Yaskawa INFORM job: demo_21_12_2023_planes_program.JBI

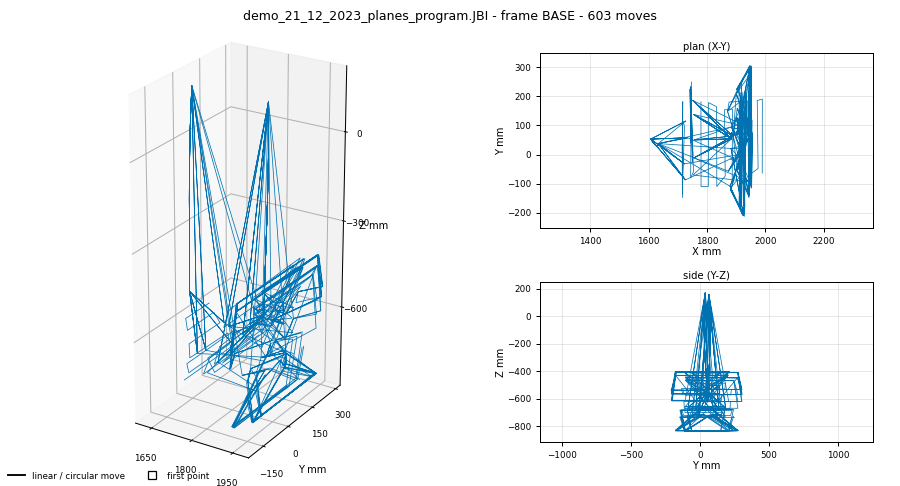
[picture p0: tool path of demo_21_12_2023_planes_program.JBI in frame BASE, 603 of 622 moves have a stored position in this frame; points joined in program order, loops and branches not executed]
/JOB
//NAME demo_21_12_2023_planes_program
//POS
///NPOS 616,0,616,0,0,0
///TOOL 0
///POSTYPE BASE
///RECTAN
///RCONF 0,0,0,0,0,0,0,0,0,0,0,0,0,0,0,0,0,0,0,0,0,0,0,0
C00000=1907.033318,105.448562,-531.357100,175.000000,-89.559174,-5.000000
C00001=1954.483034,118.521309,-531.351102,-175.000000,-89.985238,-46.086947
C00002=1951.789589,-60.582177,-405.692341,-175.000000,-58.956246,33.554175
C00003=1950.891473,275.514781,-409.751002,175.000000,-60.779903,-37.214964
C00004=1950.739483,304.407695,-531.280759,-175.000000,-89.985238,-46.086947
C00005=1904.555206,228.496419,-531.310537,175.000000,-9000000,5.000000
C00006=1955.420788,71.957040,-531.368723,175.000000,-89.985238,-46.086947
C00007=1952.438991,-107.141483,-443.395354,175.000000,-58.956472,33.555545
C00008=1950.674715,271.761571,-447.437042,-175.000000,-60.779789,-37.213566
C00009=1950.815178,300.649067,-531.282181,175.000000,-89.985238,-46.086947
C00010=1904.555206,228.496419,-531.310537,175.000000,-9000000,5.000000
C00011=1955.560862,65.001669,-531.371355,175.000000,-89.985238,-46.086947
C00012=1952.862971,-114.102374,-406.302816,-175.000000,-58.956353,33.554309
C00013=1950.927845,273.475107,-410.342085,175.000000,-60.780048,-37.215010
C00014=1950.780573,302.367348,-531.281531,175.000000,-89.985238,-46.086947
C00015=1904.555206,228.496419,-531.310537,175.000000,-9000000,5.000000
C00016=1900.400389,222.474608,-568.500057,175.000000,-89.559174,-5.000000
C00017=1947.081445,305.285270,-568.478734,-175.000000,-89.990197,-46.567779
C00018=1947.250662,275.979199,-409.311487,175.000000,-60.601810,-37.547371
C00019=1943.764744,-60.153943,-406.108555,175.000000,-59.166964,33.242469
C00020=1947.704549,119.398883,-568.525070,175.000000,-89.990197,-46.567779
C00021=1900.913317,69.456215,-568.538199,175.000000,-9000000,5.000000
C00022=1947.094044,301.526641,-568.479671,175.000000,-89.990197,-46.567779
C00023=1946.974018,272.228543,-446.996811,175.000000,-60.601591,-37.547423
C00024=1943.630528,-106.710862,-443.805636,175.000000,-59.167227,33.242548
C00025=1947.860635,72.834614,-568.536677,175.000000,-89.990197,-46.567779
C00026=1900.913317,69.456215,-568.538199,175.000000,-9000000,5.000000
C00027=1947.088284,303.244923,-568.479242,-175.000000,-89.990197,-46.567779
C00028=1947.253324,273.939620,-409.902004,-175.000000,-60.601821,-37.547527
C00029=1943.938758,-113.673732,-406.712292,175.000000,-59.167149,33.242355
C00030=1947.883950,65.879243,-568.538410,175.000000,-89.990197,-46.567779
C00031=1900.913317,69.456215,-568.538199,175.000000,-9000000,5.000000
C00032=1947.181211,275.522780,-568.486153,175.000000,-89.990197,-46.567779
C00033=1946.900224,246.230934,-467.867787,175.000000,-60.602079,-37.547614
C00034=1943.466507,-105.922888,-464.668327,175.000000,-59.167008,33.241936
C00035=1947.858017,73.615805,-568.536482,175.000000,-89.990197,-46.567779
C00036=1900.913317,69.456215,-568.538199,175.000000,-9000000,5.000000
C00037=1889.556234,63.921597,158.246462,-12.170215,-10.697646,-175.000000
C00038=1889.623159,63.877828,158.302867,-12.170828,-10.698957,-175.000000
C00039=1887.716063,68.814383,78.786651,-10.416760,-13.956672,-175.000000
C00040=1886.079895,71.876277,1.464639,-8.880031,-17.287043,-175.000000
C00041=1884.307478,73.313181,-73.802853,-7.558614,-20.681301,-175.000000
C00042=1882.911392,73.396272,-147.225748,-6.476440,-24.117963,-175.000000
C00043=1881.789821,72.259721,-218.453619,-5.660340,-27.576620,-175.000000
C00044=1880.837059,70.160415,-287.739273,5.000000,-31.424829,172.739336
C00045=1880.593414,67.184315,-355.151365,5.000000,-34.810443,174.015393
C00046=1880.906153,63.376292,-421.003543,5.000000,-38.223195,174.604447
C00047=1881.751155,59.024234,-485.031840,5.000000,-41.626153,174.627532
C00048=1883.567861,53.969547,-547.634242,5.000000,-44.999700,174.201251
C00049=1755.822095,50.404704,-618.581704,175.000000,-9000000,5.000000
C00050=1889.556234,63.921597,158.246462,-12.170215,-10.697646,-175.000000
C00051=1889.623159,63.877828,158.302867,-12.170828,-10.698957,-175.000000
C00052=1887.716063,68.814383,78.786651,-10.416760,-13.956672,-175.000000
C00053=1886.079895,71.876277,1.464639,-8.880031,-17.287043,-175.000000
C00054=1884.307478,73.313181,-73.802853,-7.558614,-20.681301,-175.000000
C00055=1882.911392,73.396272,-147.225748,-6.476440,-24.117963,-175.000000
C00056=1881.789821,72.259721,-218.453619,-5.660340,-27.576620,-175.000000
C00057=1880.837059,70.160415,-287.739273,5.000000,-31.424829,172.739336
C00058=1880.593414,67.184315,-355.151365,5.000000,-34.810443,174.015393
C00059=1880.906153,63.376292,-421.003543,5.000000,-38.223195,174.604447
C00060=1881.751155,59.024234,-485.031840,5.000000,-41.626153,174.627532
C00061=1883.567861,53.969547,-547.634242,5.000000,-44.999700,174.201251
C00062=1755.822095,50.404704,-618.581704,175.000000,-9000000,5.000000
C00063=1889.556234,63.921597,158.246462,-12.170215,-10.697646,-175.000000
C00064=1889.623159,63.877828,158.302867,-12.170828,-10.698957,-175.000000
C00065=1887.716063,68.814383,78.786651,-10.416760,-13.956672,-175.000000
C00066=1886.079895,71.876277,1.464639,-8.880031,-17.287043,-175.000000
C00067=1884.307478,73.313181,-73.802853,-7.558614,-20.681301,-175.000000
C00068=1882.911392,73.396272,-147.225748,-6.476440,-24.117963,-175.000000
C00069=1881.789821,72.259721,-218.453619,-5.660340,-27.576620,-175.000000
C00070=1880.837059,70.160415,-287.739273,5.000000,-31.424829,172.739336
C00071=1880.593414,67.184315,-355.151365,5.000000,-34.810443,174.015393
C00072=1880.906153,63.376292,-421.003543,5.000000,-38.223195,174.604447
C00073=1881.751155,59.024234,-485.031840,5.000000,-41.626153,174.627532
C00074=1883.567861,53.969547,-547.634242,5.000000,-44.999700,174.201251
C00075=1755.822095,50.404704,-618.581704,175.000000,-9000000,5.000000
C00076=1951.369555,117.933153,-618.544705,175.000000,-89.981843,-45.753303
C00077=1950.408580,-60.871163,-405.345417,-175.000000,-58.807688,33.768810
C00078=1946.465369,275.184802,-409.998652,175.000000,-60.901627,-36.982641
C00079=1945.459620,303.819540,-618.457694,175.000000,-89.981843,-45.753303
C00080=1900.287093,207.836706,-618.503937,175.000000,-9000000,5.000000
C00081=1952.849985,71.368885,-618.566501,175.000000,-89.981843,-45.753303
C00082=1951.598144,-107.427747,-443.052619,175.000000,-58.807922,33.768719
C00083=1946.295789,271.434354,-447.684920,175.000000,-60.901461,-36.982782
C00084=1945.579119,30060912,-618.459453,-175.000000,-89.981843,-45.753303
C00085=1900.287093,207.836706,-618.503937,175.000000,-9000000,5.000000
C00086=1953.071119,64.413513,-618.569757,-175.000000,-89.981843,-45.753303
C00087=1952.104538,-114.390894,-405.960815,175.000000,-58.807853,33.768670
C00088=1946.526026,273.145173,-410.589561,175.000000,-60.901614,-36.982778
C00089=1945.524489,301.779193,-618.458649,-175.000000,-89.981843,-45.753303
C00090=1900.287093,207.836706,-618.503937,175.000000,-9000000,5.000000
C00091=1952.825149,72.150076,-618.566135,-175.000000,-89.981843,-45.753303
C00092=1951.412479,-106.640599,-463.915398,175.000000,-58.807817,33.768501
C00093=1946.962416,245.436524,-468.560719,-175.000000,-60.901568,-36.983014
C00094=1946.405867,274.057050,-618.471626,175.000000,-89.981843,-45.753303
C00095=1900.287093,207.836706,-618.503937,175.000000,-9000000,5.000000
C00096=1889.556234,63.921597,158.246462,-12.170215,-10.697646,-175.000000
C00097=1889.623159,63.877828,158.302867,-12.170828,-10.698957,-175.000000
C00098=1887.716063,68.814383,78.786651,-10.416760,-13.956672,-175.000000
C00099=1886.079895,71.876277,1.464639,-8.880031,-17.287043,-175.000000
C00100=1884.307478,73.313181,-73.802853,-7.558614,-20.681301,-175.000000
C00101=1882.911392,73.396272,-147.225748,-6.476440,-24.117963,-175.000000
C00102=1881.789821,72.259721,-218.453619,-5.660340,-27.576620,-175.000000
C00103=1880.837059,70.160415,-287.739273,5.000000,-31.424829,172.739336
C00104=1880.593414,67.184315,-355.151365,5.000000,-34.810443,174.015393
C00105=1880.906153,63.376292,-421.003543,5.000000,-38.223195,174.604447
C00106=1881.751155,59.024234,-485.031840,5.000000,-41.626153,174.627532
C00107=1883.567861,53.969547,-547.634242,5.000000,-44.999700,174.201251
C00108=1750.649215,186.057193,-668.513072,175.000000,-9000000,5.000000
C00109=1889.556234,63.921597,158.246462,-12.170215,-10.697646,-175.000000
C00110=1889.623159,63.877828,158.302867,-12.170828,-10.698957,-175.000000
C00111=1887.716063,68.814383,78.786651,-10.416760,-13.956672,-175.000000
C00112=1886.079895,71.876277,1.464639,-8.880031,-17.287043,-175.000000
C00113=1884.307478,73.313181,-73.802853,-7.558614,-20.681301,-175.000000
C00114=1882.911392,73.396272,-147.225748,-6.476440,-24.117963,-175.000000
C00115=1881.789821,72.259721,-218.453619,-5.660340,-27.576620,-175.000000
C00116=1880.837059,70.160415,-287.739273,5.000000,-31.424829,172.739336
C00117=1880.593414,67.184315,-355.151365,5.000000,-34.810443,174.015393
C00118=1880.906153,63.376292,-421.003543,5.000000,-38.223195,174.604447
C00119=1881.751155,59.024234,-485.031840,5.000000,-41.626153,174.627532
C00120=1883.567861,53.969547,-547.634242,5.000000,-44.999700,174.201251
C00121=1750.649215,186.057193,-668.513072,175.000000,-9000000,5.000000
C00122=1889.556234,63.921597,158.246462,-12.170215,-10.697646,-175.000000
C00123=1889.623159,63.877828,158.302867,-12.170828,-10.698957,-175.000000
C00124=1887.716063,68.814383,78.786651,-10.416760,-13.956672,-175.000000
C00125=1886.079895,71.876277,1.464639,-8.880031,-17.287043,-175.000000
C00126=1884.307478,73.313181,-73.802853,-7.558614,-20.681301,-175.000000
C00127=1882.911392,73.396272,-147.225748,-6.476440,-24.117963,-175.000000
C00128=1881.789821,72.259721,-218.453619,-5.660340,-27.576620,-175.000000
C00129=1880.837059,70.160415,-287.739273,5.000000,-31.424829,172.739336
C00130=1880.593414,67.184315,-355.151365,5.000000,-34.810443,174.015393
C00131=1880.906153,63.376292,-421.003543,5.000000,-38.223195,174.604447
C00132=1881.751155,59.024234,-485.031840,5.000000,-41.626153,174.627532
C00133=1883.567861,53.969547,-547.634242,5.000000,-44.999700,174.201251
C00134=1750.649215,186.057193,-668.513072,175.000000,-9000000,5.000000
C00135=1941.739433,91.872264,-668.550173,5.000000,-89.981105,-135.836022
C00136=1942.819913,274.976952,-83002340,5.000000,-61.062899,143.242003
C00137=1946.018919,-60.273090,-834.731809,5.000000,-59.014144,-146.590892
C00138=1947.112174,-94.014122,-668.633050,5.000000,-89.981105,-135.836022
C00139=1905.452963,2.399975,-668.591073,175.000000,-9000000,5.000000
C00140=1941.848070,88.113636,-668.551849,5.000000,-89.981105,-135.836022
C00141=1945.998331,271.516439,-447.613467,175.000000,-60.871590,-37.040266
C00142=1950.423675,-107.356915,-443.127134,175.000000,-58.844853,33.715766
C00143=1951.553207,71.531040,-668.559002,-175.000000,-89.982681,-45.836017
C00144=1905.452963,2.399975,-668.591073,175.000000,-9000000,5.000000
C00145=1941.798406,89.831917,-668.551082,5.000000,-89.981105,-135.836022
C00146=1942.883974,272.936882,-829.346203,5.000000,-61.062928,143.241973
C00147=1947.570821,-113.793308,-834.098604,-5.000000,-59.014182,-146.590868
C00148=1951.754240,64.575669,-668.562103,-175.000000,-89.982681,-45.836017
C00149=1905.452963,2.399975,-668.591073,175.000000,-9000000,5.000000
C00150=1945.694838,274.219206,-668.468633,-175.000000,-89.982681,-45.836017
C00151=1946.589980,245.518494,-468.488538,-175.000000,-60.871631,-37.040464
C00152=1950.239929,-106.569854,-463.990120,175.000000,-58.844834,33.715560
C00153=1951.530628,72.312231,-668.558654,-175.000000,-89.982681,-45.836017
C00154=1905.452963,2.399975,-668.591073,175.000000,-9000000,5.000000
C00155=1889.556234,63.921597,158.246462,-12.170215,-10.697646,-175.000000
C00156=1889.623159,63.877828,158.302867,-12.170828,-10.698957,-175.000000
C00157=1887.716063,68.814383,78.786651,-10.416760,-13.956672,-175.000000
C00158=1886.079895,71.876277,1.464639,-8.880031,-17.287043,-175.000000
C00159=1884.307478,73.313181,-73.802853,-7.558614,-20.681301,-175.000000
C00160=1882.911392,73.396272,-147.225748,-6.476440,-24.117963,-175.000000
C00161=1881.789821,72.259721,-218.453619,-5.660340,-27.576620,-175.000000
C00162=1880.837059,70.160415,-287.739273,5.000000,-31.424829,172.739336
C00163=1880.593414,67.184315,-355.151365,5.000000,-34.810443,174.015393
C00164=1880.906153,63.376292,-421.003543,5.000000,-38.223195,174.604447
C00165=1881.751155,59.024234,-485.031840,5.000000,-41.626153,174.627532
C00166=1883.567861,53.969547,-547.634242,5.000000,-44.999700,174.201251
C00167=1754.643051,-11.429649,-718.589414,175.000000,-9000000,5.000000
C00168=1889.556234,63.921597,158.246462,-12.170215,-10.697646,-175.000000
C00169=1889.623159,63.877828,158.302867,-12.170828,-10.698957,-175.000000
C00170=1887.716063,68.814383,78.786651,-10.416760,-13.956672,-175.000000
C00171=1886.079895,71.876277,1.464639,-8.880031,-17.287043,-175.000000
C00172=1884.307478,73.313181,-73.802853,-7.558614,-20.681301,-175.000000
C00173=1882.911392,73.396272,-147.225748,-6.476440,-24.117963,-175.000000
C00174=1881.789821,72.259721,-218.453619,-5.660340,-27.576620,-175.000000
C00175=1880.837059,70.160415,-287.739273,5.000000,-31.424829,172.739336
C00176=1880.593414,67.184315,-355.151365,5.000000,-34.810443,174.015393
C00177=1880.906153,63.376292,-421.003543,5.000000,-38.223195,174.604447
C00178=1881.751155,59.024234,-485.031840,5.000000,-41.626153,174.627532
C00179=1883.567861,53.969547,-547.634242,5.000000,-44.999700,174.201251
C00180=1754.643051,-11.429649,-718.589414,175.000000,-9000000,5.000000
C00181=1889.556234,63.921597,158.246462,-12.170215,-10.697646,-175.000000
C00182=1889.623159,63.877828,158.302867,-12.170828,-10.698957,-175.000000
C00183=1887.716063,68.814383,78.786651,-10.416760,-13.956672,-175.000000
C00184=1886.079895,71.876277,1.464639,-8.880031,-17.287043,-175.000000
C00185=1884.307478,73.313181,-73.802853,-7.558614,-20.681301,-175.000000
C00186=1882.911392,73.396272,-147.225748,-6.476440,-24.117963,-175.000000
C00187=1881.789821,72.259721,-218.453619,-5.660340,-27.576620,-175.000000
C00188=1880.837059,70.160415,-287.739273,5.000000,-31.424829,172.739336
C00189=1880.593414,67.184315,-355.151365,5.000000,-34.810443,174.015393
C00190=1880.906153,63.376292,-421.003543,5.000000,-38.223195,174.604447
C00191=1881.751155,59.024234,-485.031840,5.000000,-41.626153,174.627532
C00192=1883.567861,53.969547,-547.634242,5.000000,-44.999700,174.201251
C00193=1754.643051,-11.429649,-718.589414,175.000000,-9000000,5.000000
C00194=1945.109419,-92.763747,-718.608360,5.000000,-89.988712,-136.492236
C00195=1944.744831,-59.705754,-834.062988,5.000000,-59.310215,-147.008189
C00196=1947.521106,275.607521,-830.600257,5.000000,-60.814495,142.793100
C00197=1943.996119,93.122640,-718.558252,5.000000,-89.988712,-136.492236
C00198=1903.328616,157.105618,-718.541637,175.000000,-9000000,5.000000
C00199=1950.912528,72.732070,-718.563642,-175.000000,-89.989413,-46.492234
C00200=1945.018194,-106.270873,-834.806367,-5.000000,-59.310282,-147.008065
C00201=1947.537237,271.848413,-831.332199,5.000000,-60.814515,142.793257
C00202=1944.018630,89.364012,-718.559266,-5.000000,-89.988712,-136.492236
C00203=1903.328616,157.105618,-718.541637,175.000000,-9000000,5.000000
C00204=1950.954184,65.776698,-718.565517,175.000000,-89.989413,-46.492234
C00205=1945.069512,-113.225825,-833.420115,5.000000,-59.310354,-147.008282
C00206=1947.538175,273.567484,-829.943731,5.000000,-60.814536,142.793056
C00207=1944.008339,91.082293,-718.558802,5.000000,-89.988712,-136.492236
C00208=1903.328616,157.105618,-718.541637,175.000000,-9000000,5.000000
C00209=1950.907849,73.513261,-718.563432,-175.000000,-89.989413,-46.492234
C00210=1945.021973,-105.488764,-833.644297,5.000000,-59.310234,-147.008242
C00211=1947.702278,245.845502,-830.177084,5.000000,-60.814585,142.793096
C00212=1944.174371,63.360150,-718.566275,5.000000,-89.988712,-136.492236
C00213=1903.328616,157.105618,-718.541637,175.000000,-9000000,5.000000
C00214=1889.556234,63.921597,158.246462,-12.170215,-10.697646,-175.000000
C00215=1889.623159,63.877828,158.302867,-12.170828,-10.698957,-175.000000
C00216=1887.716063,68.814383,78.786651,-10.416760,-13.956672,-175.000000
C00217=1886.079895,71.876277,1.464639,-8.880031,-17.287043,-175.000000
C00218=1884.307478,73.313181,-73.802853,-7.558614,-20.681301,-175.000000
C00219=1882.911392,73.396272,-147.225748,-6.476440,-24.117963,-175.000000
C00220=1881.789821,72.259721,-218.453619,-5.660340,-27.576620,-175.000000
C00221=1880.837059,70.160415,-287.739273,5.000000,-31.424829,172.739336
C00222=1880.593414,67.184315,-355.151365,5.000000,-34.810443,174.015393
C00223=1880.906153,63.376292,-421.003543,5.000000,-38.223195,174.604447
C00224=1881.751155,59.024234,-485.031840,5.000000,-41.626153,174.627532
C00225=1883.567861,53.969547,-547.634242,5.000000,-44.999700,174.201251
C00226=1754.303875,137.531750,-681.952455,175.000000,-9000000,5.000000
C00227=1889.556234,63.921597,158.246462,-12.170215,-10.697646,-175.000000
C00228=1889.623159,63.877828,158.302867,-12.170828,-10.698957,-175.000000
C00229=1887.716063,68.814383,78.786651,-10.416760,-13.956672,-175.000000
C00230=1886.079895,71.876277,1.464639,-8.880031,-17.287043,-175.000000
C00231=1884.307478,73.313181,-73.802853,-7.558614,-20.681301,-175.000000
C00232=1882.911392,73.396272,-147.225748,-6.476440,-24.117963,-175.000000
C00233=1881.789821,72.259721,-218.453619,-5.660340,-27.576620,-175.000000
C00234=1880.837059,70.160415,-287.739273,5.000000,-31.424829,172.739336
C00235=1880.593414,67.184315,-355.151365,5.000000,-34.810443,174.015393
C00236=1880.906153,63.376292,-421.003543,5.000000,-38.223195,174.604447
C00237=1881.751155,59.024234,-485.031840,5.000000,-41.626153,174.627532
C00238=1883.567861,53.969547,-547.634242,5.000000,-44.999700,174.201251
C00239=1754.303875,137.531750,-681.952455,175.000000,-9000000,5.000000
C00240=1889.556234,63.921597,158.246462,-12.170215,-10.697646,-175.000000
C00241=1889.623159,63.877828,158.302867,-12.170828,-10.698957,-175.000000
C00242=1887.716063,68.814383,78.786651,-10.416760,-13.956672,-175.000000
C00243=1886.079895,71.876277,1.464639,-8.880031,-17.287043,-175.000000
C00244=1884.307478,73.313181,-73.802853,-7.558614,-20.681301,-175.000000
C00245=1882.911392,73.396272,-147.225748,-6.476440,-24.117963,-175.000000
C00246=1881.789821,72.259721,-218.453619,-5.660340,-27.576620,-175.000000
C00247=1880.837059,70.160415,-287.739273,5.000000,-31.424829,172.739336
C00248=1880.593414,67.184315,-355.151365,5.000000,-34.810443,174.015393
C00249=1880.906153,63.376292,-421.003543,5.000000,-38.223195,174.604447
C00250=1881.751155,59.024234,-485.031840,5.000000,-41.626153,174.627532
C00251=1883.567861,53.969547,-547.634242,5.000000,-44.999700,174.201251
C00252=1754.303875,137.531750,-681.952455,175.000000,-9000000,5.000000
C00253=1889.556234,63.921597,158.246462,-12.170215,-10.697646,-175.000000
C00254=1889.623159,63.877828,158.302867,-12.170828,-10.698957,-175.000000
C00255=1887.716063,68.814383,78.786651,-10.416760,-13.956672,-175.000000
C00256=1886.079895,71.876277,1.464639,-8.880031,-17.287043,-175.000000
C00257=1884.307478,73.313181,-73.802853,-7.558614,-20.681301,-175.000000
C00258=1882.911392,73.396272,-147.225748,-6.476440,-24.117963,-175.000000
C00259=1881.789821,72.259721,-218.453619,-5.660340,-27.576620,-175.000000
C00260=1880.837059,70.160415,-287.739273,5.000000,-31.424829,172.739336
C00261=1880.593414,67.184315,-355.151365,5.000000,-34.810443,174.015393
C00262=1880.906153,63.376292,-421.003543,5.000000,-38.223195,174.604447
C00263=1881.751155,59.024234,-485.031840,5.000000,-41.626153,174.627532
C00264=1883.567861,53.969547,-547.634242,5.000000,-44.999700,174.201251
C00265=1754.303875,137.531750,-681.952455,175.000000,-9000000,5.000000
C00266=1944.740157,93.554557,-681.959370,-5.000000,-89.991235,-136.713417
C00267=1949.343284,275.815144,-830.807048,5.000000,-60.729125,142.642519
C00268=1944.552036,-59.508291,-833.842699,-5.000000,-59.408325,-147.150251
C00269=1944.418269,-92.331830,-681.998435,5.000000,-89.991235,-136.713417
C00270=1903.729498,-56.819837,-681.991470,175.000000,-9000000,5.000000
C00271=1944.733648,89.795928,-681.960160,5.000000,-89.991235,-136.713417
C00272=1949.330371,272.055939,-831.538811,5.000000,-60.729126,142.642723
C00273=1944.465133,-106.073368,-834.582953,5.000000,-59.408549,-147.150209
C00274=1944.337637,-138.896099,-682.008221,5.000000,-89.991235,-136.713417
C00275=1903.729498,-56.819837,-681.991470,175.000000,-9000000,5.000000
C00276=1944.736623,91.514210,-681.959798,5.000000,-89.991235,-136.713417
C00277=1949.344074,273.774978,-830.150143,5.000000,-60.729278,142.642595
C00278=1944.463820,-113.028499,-833.196650,-5.000000,-59.408464,-147.150271
C00279=1944.325592,-145.851470,-682.009683,-5.000000,-89.991235,-136.713417
C00280=1903.729498,-56.819837,-681.991470,175.000000,-9000000,5.000000
C00281=1944.688619,63.792067,-681.965625,5.000000,-89.991235,-136.713417
C00282=1949.294155,246.053003,-830.381801,5.000000,-60.729348,142.642640
C00283=1944.476511,-105.291509,-833.421558,-5.000000,-59.408226,-147.150148
C00284=1944.338989,-138.114908,-682.008057,-5.000000,-89.991235,-136.713417
C00285=1903.729498,-56.819837,-681.991470,175.000000,-9000000,5.000000
C00286=1889.556234,63.921597,158.246462,-12.170215,-10.697646,-175.000000
C00287=1889.623159,63.877828,158.302867,-12.170828,-10.698957,-175.000000
C00288=1887.716063,68.814383,78.786651,-10.416760,-13.956672,-175.000000
C00289=1886.079895,71.876277,1.464639,-8.880031,-17.287043,-175.000000
C00290=1884.307478,73.313181,-73.802853,-7.558614,-20.681301,-175.000000
C00291=1882.911392,73.396272,-147.225748,-6.476440,-24.117963,-175.000000
C00292=1881.789821,72.259721,-218.453619,-5.660340,-27.576620,-175.000000
C00293=1880.837059,70.160415,-287.739273,5.000000,-31.424829,172.739336
C00294=1880.593414,67.184315,-355.151365,5.000000,-34.810443,174.015393
C00295=1880.906153,63.376292,-421.003543,5.000000,-38.223195,174.604447
C00296=1881.751155,59.024234,-485.031840,5.000000,-41.626153,174.627532
C00297=1883.567861,53.969547,-547.634242,5.000000,-44.999700,174.201251
C00298=1752.029754,-69.858282,-731.982788,175.000000,-9000000,5.000000
C00299=1942.290332,-92.571429,-731.985649,5.000000,-89.989735,-136.581685
C00300=1942.741090,-59.625904,-833.959304,5.000000,-59.349806,-147.065680
C00301=1946.332931,275.692102,-830.669243,5.000000,-60.779904,142.731914
C00302=1941.757450,93.314957,-731.940007,5.000000,-89.989735,-136.581685
C00303=1901.186698,127.297726,-731.932241,175.000000,-9000000,5.000000
C00304=1942.423818,-139.135698,-731.997082,-5.000000,-89.989735,-136.581685
C00305=1942.867588,-106.191308,-834.700067,5.000000,-59.350536,-147.065659
C00306=1946.336088,271.931920,-831.400871,5.000000,-60.780021,142.732704
C00307=1941.768225,89.556329,-731.940930,5.000000,-89.989735,-136.581685
C00308=1901.186698,127.297726,-731.932241,175.000000,-9000000,5.000000
C00309=1942.443758,-146.091069,-731.998790,5.000000,-89.989735,-136.581685
C00310=1942.898325,-113.146105,-833.314387,5.000000,-59.350283,-147.065833
C00311=1946.341642,273.651504,-83011340,-5.000000,-60.780524,142.732427
C00312=1941.763299,91.274610,-731.940508,5.000000,-89.989735,-136.581685
C00313=1901.186698,127.297726,-731.932241,175.000000,-9000000,5.000000
C00314=1942.421579,-138.354507,-731.996890,5.000000,-89.989735,-136.581685
C00315=1942.874857,-105.408541,-833.539318,5.000000,-59.349912,-147.065963
C00316=1946.420644,245.930307,-830.244454,5.000000,-60.780388,142.731955
C00317=1941.842770,63.552467,-731.947315,5.000000,-89.989735,-136.581685
C00318=1901.186698,127.297726,-731.932241,18000000,-6000000,000000
C00319=1744.163168,103.731386,-533.824639,5.000000,-89.520571,175.000000
C00320=174053701,229.900913,-533.872980,5.000000,-89.520571,175.000000
C00321=1740.139661,223.998415,-571.035053,5.000000,-89.520571,175.000000
C00322=1745.940022,70.141244,-570.969500,5.000000,-89.520571,175.000000
C00323=1743.699231,39.699755,-620.986636,5.000000,-89.520571,175.000000
C00324=1743.736408,220.431312,-621.006311,5.000000,-89.520571,175.000000
C00325=1743.938875,217.744936,-671.006071,5.000000,-89.520571,175.000000
C00326=1751.483237,3.541384,-670.919251,5.000000,-89.520571,175.000000
C00327=1749.639439,-25.239911,-720.933248,5.000000,-89.520571,175.000000
C00328=1742.908909,221.089212,-721.016811,5.000000,-89.520571,175.000000
C00329=1744.116223,233.211429,-684.407259,5.000000,-89.520571,175.000000
C00330=1753.513039,-58.753955,-684.296338,5.000000,-89.520571,175.000000
C00331=1743.842593,-79.925565,-734.376670,5.000000,-89.520571,175.000000
C00332=1746.666835,248.969851,-734.389409,18000000,-6000000,000000
C00333=1717.090387,-3.043329,-525.112751,-5.000000,-89.896397,-175.000000
C00334=1715.582850,-134.626368,-525.110413,-5.000000,-89.896397,-175.000000
C00335=1715.652100,-125.400738,-569.935144,-5.000000,-89.896397,-175.000000
C00336=1714.677180,27.356629,-569.942784,-5.000000,-89.896397,-175.000000
C00337=1716.200893,60.962231,-619.941404,-5.000000,-89.896397,-175.000000
C00338=1715.751699,-117.347731,-619.935355,-5.000000,-89.896397,-175.000000
C00339=1715.928918,-113.952816,-669.935247,-5.000000,-89.896397,-175.000000
C00340=1722.693836,97.479027,-669.931151,-5.000000,-89.896397,-175.000000
C00341=1715.897617,118.196967,-719.944318,-5.000000,-89.896397,-175.000000
C00342=1715.387537,-119.836296,-719.936081,-5.000000,-89.896397,-175.000000
C00343=1715.633277,-131.036930,-683.332748,-5.000000,-89.896397,-175.000000
C00344=1716.169223,154.077841,-683.342749,-5.000000,-89.896397,-175.000000
C00345=1716.790282,181.476308,-733.342762,-5.000000,-89.896397,-175.000000
C00346=1716.082413,-146.810235,-733.331410,18000000,-6000000,000000
C00347=1878.651480,-14.855522,-537.062852,175.000000,-88.097363,-5.000000
C00348=1922.281376,-31.606783,-537.075471,5.000000,-89.970325,-133.774897
C00349=1921.565087,150.704793,-403.442618,-175.000000,-59.777968,-34.809520
C00350=193001845,-180.972615,-402.864288,175.000000,-59.463968,37.005505
C00351=1927.472959,-211.533153,-537.206326,5.000000,-89.970325,-133.774897
C00352=1881.720340,-121.213359,-537.140203,-175.000000,-89.999999,5.000000
C00353=1920.818604,19.088977,-537.038602,5.000000,-89.970325,-133.774897
C00354=1919.228609,201.394910,-429.719115,175.000000,-59.777914,-34.809652
C00355=1929.050258,-178.319874,-429.176665,-175.000000,-59.464338,37.005437
C00356=1927.396225,-208.873762,-537.204392,5.000000,-89.970325,-133.774897
C00357=1881.720340,-121.213359,-537.140203,-175.000000,-89.999999,5.000000
C00358=1920.513394,29.666722,-537.030909,5.000000,-89.970325,-133.774897
C00359=1919.781998,211.979285,-403.878868,-175.000000,-59.777995,-34.809835
C00360=1929.779916,-173.832647,-403.339775,175.000000,-59.463942,37.005472
C00361=1927.266945,-204.393259,-537.201133,5.000000,-89.970325,-133.774897
C00362=1881.720340,-121.213359,-537.140203,-175.000000,-89.999999,5.000000
C00363=1880.324864,-121.388096,-563.848788,175.000000,-88.097363,-5.000000
C00364=1924.477331,-209.309200,-563.788106,175.000000,-89.972614,45.007217
C00365=1928.547064,-179.814548,-403.922550,175.000000,-59.929655,36.165405
C00366=1930.987541,151.882666,-402.634194,-175.000000,-59.304595,-35.645060
C00367=1926.936425,-29.382830,-563.911404,-175.000000,-89.972614,45.007217
C00368=1882.272046,21.082740,-563.946419,-175.000000,-89.999999,5.000000
C00369=1924.513677,-206.649809,-563.789928,175.000000,-89.972614,45.007217
C00370=1927.708515,-177.161618,-430.238366,175.000000,-59.929885,36.165300
C00371=1930.807006,202.572899,-428.982251,175.000000,-59.304515,-35.645269
C00372=1927.629296,21.312930,-563.946144,-175.000000,-89.972614,45.007217
C00373=1882.272046,21.082740,-563.946419,-175.000000,-89.999999,5.000000
C00374=1924.574913,-202.169306,-563.792998,175.000000,-89.972614,45.007217
C00375=1928.629244,-172.674803,-404.407974,-175.000000,-59.929560,36.165524
C00376=1931.808346,213.156570,-403.157323,175.000000,-59.304780,-35.644990
C00377=1927.773864,31.890675,-563.953393,-175.000000,-89.972614,45.007217
C00378=1882.272046,21.082740,-563.946419,-175.000000,-89.999999,5.000000
C00379=1632.892026,37.747570,168.285511,11.376794,11.539120,-175.000000
C00380=1632.827507,37.791596,168.344749,11.377310,11.540473,-175.000000
C00381=1631.070965,33.437366,89.156599,9.359774,14.678599,-175.000000
C00382=1629.142714,30.961716,12.173907,7.532522,17.899912,-175.000000
C00383=1627.447598,30.112422,-62.761067,5.887863,21.196066,-175.000000
C00384=1625.471635,30.613173,-135.840164,5.000000,24.547751,-175.000000
C00385=1623.335953,32.324503,-206.720523,5.000000,27.937078,-175.000000
C00386=1621.140462,34.985091,-275.661674,5.000000,-31.424829,-5.000000
C00387=1618.347384,38.503638,-342.713252,5.000000,-34.810443,-5.000000
C00388=1615.097741,42.831038,-408.197316,-5.000000,-38.223195,-5.000000
C00389=1611.433002,47.673610,-471.854532,-5.000000,-41.626153,-5.000000
C00390=1606.899024,53.186011,-534.066843,5.000000,-44.999700,-5.000000
C00391=1733.759636,57.739172,-614.031896,-175.000000,-89.999999,5.000000
C00392=1632.892026,37.747570,168.285511,11.376794,11.539120,-175.000000
C00393=1632.827507,37.791596,168.344749,11.377310,11.540473,-175.000000
C00394=1631.070965,33.437366,89.156599,9.359774,14.678599,-175.000000
C00395=1629.142714,30.961716,12.173907,7.532522,17.899912,-175.000000
C00396=1627.447598,30.112422,-62.761067,5.887863,21.196066,-175.000000
C00397=1625.471635,30.613173,-135.840164,5.000000,24.547751,-175.000000
C00398=1623.335953,32.324503,-206.720523,5.000000,27.937078,-175.000000
C00399=1621.140462,34.985091,-275.661674,5.000000,-31.424829,-5.000000
C00400=1618.347384,38.503638,-342.713252,5.000000,-34.810443,-5.000000
C00401=1615.097741,42.831038,-408.197316,-5.000000,-38.223195,-5.000000
C00402=1611.433002,47.673610,-471.854532,-5.000000,-41.626153,-5.000000
C00403=1606.899024,53.186011,-534.066843,5.000000,-44.999700,-5.000000
C00404=1733.759636,57.739172,-614.031896,-175.000000,-89.999999,5.000000
C00405=1632.892026,37.747570,168.285511,11.376794,11.539120,-175.000000
C00406=1632.827507,37.791596,168.344749,11.377310,11.540473,-175.000000
C00407=1631.070965,33.437366,89.156599,9.359774,14.678599,-175.000000
C00408=1629.142714,30.961716,12.173907,7.532522,17.899912,-175.000000
C00409=1627.447598,30.112422,-62.761067,5.887863,21.196066,-175.000000
C00410=1625.471635,30.613173,-135.840164,5.000000,24.547751,-175.000000
C00411=1623.335953,32.324503,-206.720523,5.000000,27.937078,-175.000000
C00412=1621.140462,34.985091,-275.661674,5.000000,-31.424829,-5.000000
C00413=1618.347384,38.503638,-342.713252,5.000000,-34.810443,-5.000000
C00414=1615.097741,42.831038,-408.197316,-5.000000,-38.223195,-5.000000
C00415=1611.433002,47.673610,-471.854532,-5.000000,-41.626153,-5.000000
C00416=1606.899024,53.186011,-534.066843,5.000000,-44.999700,-5.000000
C00417=1733.759636,57.739172,-614.031896,-175.000000,-89.999999,5.000000
C00418=1927.328468,-28.623634,-613.927963,175.000000,-89.953719,44.592323
C00419=1934.355931,152.264475,-402.352265,175.000000,-59.137640,-35.925997
C00420=1928.209886,-179.401451,-404.276647,-175.000000,-6082734,35.875902
C00421=1922.262476,-208.550004,-613.718064,175.000000,-89.953719,44.592323
C00422=1879.006381,-108.476117,-613.835557,-175.000000,-89.999999,5.000000
C00423=1928.755854,22.072125,-613.987103,175.000000,-89.953719,44.592323
C00424=1934.908337,202.954235,-428.725120,175.000000,-59.137750,-35.925865
C00425=1927.410838,-176.748780,-430.593291,175.000000,-6082759,35.876024
C00426=1922.337354,-205.890613,-613.721167,-175.000000,-89.953719,44.592323
C00427=1879.006381,-108.476117,-613.835557,-175.000000,-89.999999,5.000000
C00428=1929.053680,32.649871,-613.999443,175.000000,-89.953719,44.592323
C00429=1936.065735,213.538641,-402.904501,175.000000,-59.137643,-35.926149
C00430=1928.394599,-172.261419,-404.765772,175.000000,-6082764,35.875812
C00431=1922.463506,-201.410110,-613.726394,175.000000,-89.953719,44.592323
C00432=1879.006381,-108.476117,-613.835557,-175.000000,-89.999999,5.000000
C00433=1632.892026,37.747570,168.285511,11.376794,11.539120,-175.000000
C00434=1632.827507,37.791596,168.344749,11.377310,11.540473,-175.000000
C00435=1631.070965,33.437366,89.156599,9.359774,14.678599,-175.000000
C00436=1629.142714,30.961716,12.173907,7.532522,17.899912,-175.000000
C00437=1627.447598,30.112422,-62.761067,5.887863,21.196066,-175.000000
C00438=1625.471635,30.613173,-135.840164,5.000000,24.547751,-175.000000
C00439=1623.335953,32.324503,-206.720523,5.000000,27.937078,-175.000000
C00440=1621.140462,34.985091,-275.661674,5.000000,-31.424829,-5.000000
C00441=1618.347384,38.503638,-342.713252,5.000000,-34.810443,-5.000000
C00442=1615.097741,42.831038,-408.197316,-5.000000,-38.223195,-5.000000
C00443=1611.433002,47.673610,-471.854532,-5.000000,-41.626153,-5.000000
C00444=1606.899024,53.186011,-534.066843,5.000000,-44.999700,-5.000000
C00445=1726.034177,-86.452165,-663.769497,-175.000000,-89.999999,5.000000
C00446=1632.892026,37.747570,168.285511,11.376794,11.539120,-175.000000
C00447=1632.827507,37.791596,168.344749,11.377310,11.540473,-175.000000
C00448=1631.070965,33.437366,89.156599,9.359774,14.678599,-175.000000
C00449=1629.142714,30.961716,12.173907,7.532522,17.899912,-175.000000
C00450=1627.447598,30.112422,-62.761067,5.887863,21.196066,-175.000000
C00451=1625.471635,30.613173,-135.840164,5.000000,24.547751,-175.000000
C00452=1623.335953,32.324503,-206.720523,5.000000,27.937078,-175.000000
C00453=1621.140462,34.985091,-275.661674,5.000000,-31.424829,-5.000000
C00454=1618.347384,38.503638,-342.713252,5.000000,-34.810443,-5.000000
C00455=1615.097741,42.831038,-408.197316,-5.000000,-38.223195,-5.000000
C00456=1611.433002,47.673610,-471.854532,-5.000000,-41.626153,-5.000000
C00457=1606.899024,53.186011,-534.066843,5.000000,-44.999700,-5.000000
C00458=1726.034177,-86.452165,-663.769497,-175.000000,-89.999999,5.000000
C00459=1632.892026,37.747570,168.285511,11.376794,11.539120,-175.000000
C00460=1632.827507,37.791596,168.344749,11.377310,11.540473,-175.000000
C00461=1631.070965,33.437366,89.156599,9.359774,14.678599,-175.000000
C00462=1629.142714,30.961716,12.173907,7.532522,17.899912,-175.000000
C00463=1627.447598,30.112422,-62.761067,5.887863,21.196066,-175.000000
C00464=1625.471635,30.613173,-135.840164,5.000000,24.547751,-175.000000
C00465=1623.335953,32.324503,-206.720523,5.000000,27.937078,-175.000000
C00466=1621.140462,34.985091,-275.661674,5.000000,-31.424829,-5.000000
C00467=1618.347384,38.503638,-342.713252,5.000000,-34.810443,-5.000000
C00468=1615.097741,42.831038,-408.197316,-5.000000,-38.223195,-5.000000
C00469=1611.433002,47.673610,-471.854532,-5.000000,-41.626153,-5.000000
C00470=1606.899024,53.186011,-534.066843,5.000000,-44.999700,-5.000000
C00471=1726.034177,-86.452165,-663.769497,-175.000000,-89.999999,5.000000
C00472=1920.539714,4.263698,-663.911228,-5.000000,-89.932967,134.210886
C00473=1910.898002,-177.437238,-827.999831,5.000000,-61.053218,-145.607856
C00474=1920.404737,150.655474,-831.364143,5.000000,-59.702147,145.141042
C00475=1928.004667,184.190068,-664.200819,-5.000000,-89.932967,134.210886
C00476=1883.449535,94.716725,-664.057728,-175.000000,-89.999999,5.000000
C00477=1920.650049,6.923090,-663.915509,-5.000000,-89.932967,134.210886
C00478=1924.658226,-176.360358,-430.832978,175.000000,-60.221242,35.608083
C00479=1936.207328,203.296551,-428.400389,-175.000000,-58.981452,-36.182638
C00480=1927.186315,22.774189,-663.940889,175.000000,-89.936580,44.210812
C00481=1883.449535,94.716725,-664.057728,-175.000000,-89.999999,5.000000
C00482=1920.835940,11.403592,-663.922720,5.000000,-89.932967,134.210886
C00483=1911.126712,-170.297556,-83025090,-5.000000,-61.053265,-145.607951
C00484=1922.880036,211.929158,-833.476605,-5.000000,-59.702167,145.140969
C00485=1927.625174,33.351935,-663.957914,175.000000,-89.936580,44.210812
C00486=1883.449535,94.716725,-664.057728,-175.000000,-89.999999,5.000000
C00487=1632.892026,37.747570,168.285511,11.376794,11.539120,-175.000000
C00488=1632.827507,37.791596,168.344749,11.377310,11.540473,-175.000000
C00489=1631.070965,33.437366,89.156599,9.359774,14.678599,-175.000000
C00490=1629.142714,30.961716,12.173907,7.532522,17.899912,-175.000000
C00491=1627.447598,30.112422,-62.761067,5.887863,21.196066,-175.000000
C00492=1625.471635,30.613173,-135.840164,5.000000,24.547751,-175.000000
C00493=1623.335953,32.324503,-206.720523,5.000000,27.937078,-175.000000
C00494=1621.140462,34.985091,-275.661674,5.000000,-31.424829,-5.000000
C00495=1618.347384,38.503638,-342.713252,5.000000,-34.810443,-5.000000
C00496=1615.097741,42.831038,-408.197316,-5.000000,-38.223195,-5.000000
C00497=1611.433002,47.673610,-471.854532,-5.000000,-41.626153,-5.000000
C00498=1606.899024,53.186011,-534.066843,5.000000,-44.999700,-5.000000
C00499=1726.693036,114.996608,-713.865552,-175.000000,-89.999999,5.000000
C00500=1632.892026,37.747570,168.285511,11.376794,11.539120,-175.000000
C00501=1632.827507,37.791596,168.344749,11.377310,11.540473,-175.000000
C00502=1631.070965,33.437366,89.156599,9.359774,14.678599,-175.000000
C00503=1629.142714,30.961716,12.173907,7.532522,17.899912,-175.000000
C00504=1627.447598,30.112422,-62.761067,5.887863,21.196066,-175.000000
C00505=1625.471635,30.613173,-135.840164,5.000000,24.547751,-175.000000
C00506=1623.335953,32.324503,-206.720523,5.000000,27.937078,-175.000000
C00507=1621.140462,34.985091,-275.661674,5.000000,-31.424829,-5.000000
C00508=1618.347384,38.503638,-342.713252,5.000000,-34.810443,-5.000000
C00509=1615.097741,42.831038,-408.197316,-5.000000,-38.223195,-5.000000
C00510=1611.433002,47.673610,-471.854532,-5.000000,-41.626153,-5.000000
C00511=1606.899024,53.186011,-534.066843,5.000000,-44.999700,-5.000000
C00512=1726.693036,114.996608,-713.865552,-175.000000,-89.999999,5.000000
C00513=192088536,183.138293,-713.927835,5.000000,-89.960762,134.777856
C00514=1914.469398,150.182209,-830.610434,-5.000000,-59.958872,145.498573
C00515=1909.995260,-177.975773,-828.476193,5.000000,-60.821358,-145.233200
C00516=1916.188331,3.211923,-713.756664,5.000000,-89.960762,134.777856
C00517=1872.907666,-56.874190,-713.700058,-175.000000,-89.999999,5.000000
C00518=1920.364938,21.703709,-713.774206,175.000000,-89.962134,44.777830
C00519=1915.474130,200.877744,-833.502171,5.000000,-59.958839,145.498456
C00520=1909.957397,-175.317287,-831.321759,5.000000,-60.821521,-145.233339
C00521=1916.245978,5.871314,-713.759194,5.000000,-89.960762,134.777856
C00522=1872.907666,-56.874190,-713.700058,-175.000000,-89.999999,5.000000
C00523=1920.594228,32.281454,-713.784269,175.000000,-89.962134,44.777830
C00524=1915.731735,211.456180,-832.682834,-5.000000,-59.958784,145.498303
C00525=191081689,-170.835831,-830.496480,-5.000000,-60.821517,-145.233479
C00526=1916.343101,10.351817,-713.763456,5.000000,-89.960762,134.777856
C00527=1872.907666,-56.874190,-713.700058,-175.000000,-89.999999,5.000000
C00528=1632.892026,37.747570,168.285511,11.376794,11.539120,-175.000000
C00529=1632.827507,37.791596,168.344749,11.377310,11.540473,-175.000000
C00530=1631.070965,33.437366,89.156599,9.359774,14.678599,-175.000000
C00531=1629.142714,30.961716,12.173907,7.532522,17.899912,-175.000000
C00532=1627.447598,30.112422,-62.761067,5.887863,21.196066,-175.000000
C00533=1625.471635,30.613173,-135.840164,5.000000,24.547751,-175.000000
C00534=1623.335953,32.324503,-206.720523,5.000000,27.937078,-175.000000
C00535=1621.140462,34.985091,-275.661674,5.000000,-31.424829,-5.000000
C00536=1618.347384,38.503638,-342.713252,5.000000,-34.810443,-5.000000
C00537=1615.097741,42.831038,-408.197316,-5.000000,-38.223195,-5.000000
C00538=1611.433002,47.673610,-471.854532,-5.000000,-41.626153,-5.000000
C00539=1606.899024,53.186011,-534.066843,5.000000,-44.999700,-5.000000
C00540=1722.432179,-31.716582,-677.115122,-175.000000,-89.999999,5.000000
C00541=1632.892026,37.747570,168.285511,11.376794,11.539120,-175.000000
C00542=1632.827507,37.791596,168.344749,11.377310,11.540473,-175.000000
C00543=1631.070965,33.437366,89.156599,9.359774,14.678599,-175.000000
C00544=1629.142714,30.961716,12.173907,7.532522,17.899912,-175.000000
C00545=1627.447598,30.112422,-62.761067,5.887863,21.196066,-175.000000
C00546=1625.471635,30.613173,-135.840164,5.000000,24.547751,-175.000000
C00547=1623.335953,32.324503,-206.720523,5.000000,27.937078,-175.000000
C00548=1621.140462,34.985091,-275.661674,5.000000,-31.424829,-5.000000
C00549=1618.347384,38.503638,-342.713252,5.000000,-34.810443,-5.000000
C00550=1615.097741,42.831038,-408.197316,-5.000000,-38.223195,-5.000000
C00551=1611.433002,47.673610,-471.854532,-5.000000,-41.626153,-5.000000
C00552=1606.899024,53.186011,-534.066843,5.000000,-44.999700,-5.000000
C00553=1722.432179,-31.716582,-677.115122,-175.000000,-89.999999,5.000000
C00554=1632.892026,37.747570,168.285511,11.376794,11.539120,-175.000000
C00555=1632.827507,37.791596,168.344749,11.377310,11.540473,-175.000000
C00556=1631.070965,33.437366,89.156599,9.359774,14.678599,-175.000000
C00557=1629.142714,30.961716,12.173907,7.532522,17.899912,-175.000000
C00558=1627.447598,30.112422,-62.761067,5.887863,21.196066,-175.000000
C00559=1625.471635,30.613173,-135.840164,5.000000,24.547751,-175.000000
C00560=1623.335953,32.324503,-206.720523,5.000000,27.937078,-175.000000
C00561=1621.140462,34.985091,-275.661674,5.000000,-31.424829,-5.000000
C00562=1618.347384,38.503638,-342.713252,5.000000,-34.810443,-5.000000
C00563=1615.097741,42.831038,-408.197316,-5.000000,-38.223195,-5.000000
C00564=1611.433002,47.673610,-471.854532,-5.000000,-41.626153,-5.000000
C00565=1606.899024,53.186011,-534.066843,5.000000,-44.999700,-5.000000
C00566=1722.432179,-31.716582,-677.115122,-175.000000,-89.999999,5.000000
C00567=1915.883362,1.399692,-677.109901,175.000000,-89.993040,-44.253831
C00568=1914.391368,-178.853382,-829.511267,-5.000000,-60.413335,-144.601713
C00569=1910.278323,149.329618,-829.546886,5.000000,-60.384120,146.118068
C00570=1913.701168,181.326063,-677.079017,-175.000000,-89.993040,-44.253831
C00571=1870.264439,147.907785,-677.084649,-175.000000,-89.999999,5.000000
C00572=1915.851108,4.059084,-677.109444,175.000000,-89.993040,-44.253831
C00573=1914.263471,-176.194916,-832.353714,-5.000000,-60.413556,-144.601868
C00574=1909.568812,20025076,-832.381489,5.000000,-60.384173,146.118026
C00575=1913.086317,232.021822,-677.070316,175.000000,-89.993040,-44.253831
C00576=1870.264439,147.907785,-677.084649,-175.000000,-89.999999,5.000000
C00577=1915.796767,8.539586,-677.108675,-175.000000,-89.993040,-44.253831
C00578=1914.237186,-171.713611,-831.523763,5.000000,-60.413402,-144.601868
C00579=1909.468476,210.603467,-831.550117,-5.000000,-60.384183,146.117925
C00580=1912.958028,242.599568,-677.068500,-175.000000,-89.993040,-44.253831
C00581=1870.264439,147.907785,-677.084649,-175.000000,-89.999999,5.000000
C00582=1875.744531,180.347603,-727.301779,175.000000,-88.097363,-5.000000
C00583=1918.943093,181.949316,-727.302001,5.000000,-89.990941,135.406649
C00584=1916.994055,149.634481,-83090881,-5.000000,-60.236650,145.899702
C00585=1918.095090,-178.551385,-829.318448,5.000000,-60.558433,-144.822239
C00586=1918.992783,2.022946,-727.262044,5.000000,-89.990941,135.406649
C00587=1875.805406,-4082577,-727.252827,-175.000000,-89.999999,5.000000
C00588=1918.929093,232.645075,-727.313260,-5.000000,-89.990941,135.406649
C00589=1916.884577,200.329726,-832.944726,-5.000000,-60.237016,145.899895
C00590=1918.001707,-175.894247,-832.162850,5.000000,-60.558276,-144.821531
C00591=1918.992048,4.682337,-727.262634,-5.000000,-89.990941,135.406649
C00592=1875.805406,-4082577,-727.252827,-175.000000,-89.999999,5.000000
C00593=1918.926171,243.222821,-727.315609,5.000000,-89.990941,135.406649
C00594=1916.911327,210.909103,-832.118242,5.000000,-60.236717,145.899148
C00595=1918.025990,-171.411615,-831.333950,-5.000000,-60.558419,-144.822361
C00596=1918.990811,9.162840,-727.263629,5.000000,-89.990941,135.406649
C00597=1875.805406,-4082577,-727.252827,18000000,-6000000,000000
C00598=1989.146713,-63.408911,-414.613847,-175.000000,-57.317825,-5.000000
C00599=1989.481278,190.186409,-412.596769,-175.000000,-57.317825,-5.000000
C00600=1972.012521,185.428395,-447.647916,-175.000000,-57.317825,-5.000000
C00601=1974.980272,-47.365365,-451.600578,-175.000000,-57.317825,-5.000000
C00602=1942.159597,-71.671312,-490.165115,-175.000000,-57.317825,-5.000000
C00603=1939.445614,183.844710,-486.175291,-175.000000,-57.317825,-5.000000
C00604=1913.123908,180.478868,-528.724948,-175.000000,-57.317825,-5.000000
C00605=1915.291016,-72.466264,-532.341301,-175.000000,-57.317825,-5.000000
C00606=1886.227605,-107.779014,-573.413171,-175.000000,-57.317825,-5.000000
C00607=1886.895611,156.356484,-571.517200,-175.000000,-57.317825,-5.000000
C00608=1859.727942,153.368452,-613.520807,-175.000000,-57.317825,-5.000000
C00609=1862.372901,-73.234551,-617.211900,-175.000000,-57.317825,-5.000000
C00610=1833.493860,-109.096833,-658.406889,-175.000000,-57.317825,-5.000000
C00611=1832.756064,164.045975,-655.529759,-175.000000,-57.317825,-5.000000
C00612=1805.184973,178.337356,-697.122482,-175.000000,-57.317825,-5.000000
C00613=1804.387680,-109.301551,-699.142351,-175.000000,-57.317825,-5.000000
C00614=1779.535327,-109.780674,-656.006725,-175.000000,-57.317825,-5.000000
C00615=1779.101270,180.960225,-653.169586,18000000,-6000000,000000
///POSTYPE PULSE
///PULSE
EC00000=0
EC00001=0
EC00002=0
EC00003=0
EC00004=0
EC00005=0
EC00006=0
EC00007=0
EC00008=0
EC00009=0
EC00010=0
EC00011=0
EC00012=0
EC00013=0
EC00014=0
EC00015=0
EC00016=0
EC00017=0
EC00018=0
EC00019=0
EC00020=0
EC00021=0
EC00022=0
EC00023=0
EC00024=0
EC00025=0
EC00026=0
EC00027=0
EC00028=0
EC00029=0
EC00030=0
EC00031=0
EC00032=0
EC00033=0
EC00034=0
EC00035=0
EC00036=0
EC00037=0
EC00038=0
EC00039=0
EC00040=0
EC00041=0
EC00042=0
EC00043=0
EC00044=0
EC00045=0
EC00046=0
EC00047=0
EC00048=0
EC00049=0
EC00050=0
EC00051=0
EC00052=0
EC00053=0
EC00054=0
EC00055=0
EC00056=0
EC00057=0
EC00058=0
EC00059=0
EC00060=0
EC00061=0
EC00062=0
EC00063=0
EC00064=0
EC00065=0
EC00066=0
EC00067=0
EC00068=0
EC00069=0
EC00070=0
EC00071=0
EC00072=0
EC00073=0
EC00074=0
EC00075=0
EC00076=0
EC00077=0
EC00078=0
EC00079=0
EC00080=0
EC00081=0
EC00082=0
EC00083=0
EC00084=0
EC00085=0
EC00086=0
EC00087=0
EC00088=0
EC00089=0
EC00090=0
EC00091=0
EC00092=0
EC00093=0
EC00094=0
EC00095=0
EC00096=0
EC00097=0
EC00098=0
EC00099=0
EC00100=0
EC00101=0
EC00102=0
EC00103=0
EC00104=0
EC00105=0
EC00106=0
EC00107=0
EC00108=0
EC00109=0
EC00110=0
EC00111=0
EC00112=0
EC00113=0
EC00114=0
EC00115=0
EC00116=0
EC00117=0
EC00118=0
EC00119=0
EC00120=0
EC00121=0
EC00122=0
EC00123=0
EC00124=0
EC00125=0
EC00126=0
EC00127=0
EC00128=0
EC00129=0
EC00130=0
EC00131=0
EC00132=0
EC00133=0
EC00134=0
EC00135=0
EC00136=0
EC00137=0
EC00138=0
EC00139=0
EC00140=0
EC00141=0
EC00142=0
EC00143=0
EC00144=0
EC00145=0
EC00146=0
EC00147=0
EC00148=0
EC00149=0
EC00150=0
EC00151=0
EC00152=0
EC00153=0
EC00154=0
EC00155=0
EC00156=0
EC00157=0
EC00158=0
EC00159=0
EC00160=0
EC00161=0
EC00162=0
EC00163=0
EC00164=0
EC00165=0
EC00166=0
EC00167=0
EC00168=0
EC00169=0
EC00170=0
EC00171=0
EC00172=0
EC00173=0
EC00174=0
EC00175=0
EC00176=0
EC00177=0
EC00178=0
EC00179=0
EC00180=0
EC00181=0
EC00182=0
EC00183=0
EC00184=0
EC00185=0
EC00186=0
EC00187=0
EC00188=0
EC00189=0
EC00190=0
EC00191=0
EC00192=0
EC00193=0
EC00194=0
EC00195=0
EC00196=0
EC00197=0
EC00198=0
EC00199=0
EC00200=0
EC00201=0
EC00202=0
EC00203=0
EC00204=0
EC00205=0
EC00206=0
EC00207=0
EC00208=0
EC00209=0
EC00210=0
EC00211=0
EC00212=0
EC00213=0
EC00214=0
EC00215=0
EC00216=0
EC00217=0
EC00218=0
EC00219=0
EC00220=0
EC00221=0
EC00222=0
EC00223=0
EC00224=0
EC00225=0
EC00226=0
EC00227=0
EC00228=0
EC00229=0
EC00230=0
EC00231=0
EC00232=0
EC00233=0
EC00234=0
EC00235=0
EC00236=0
EC00237=0
EC00238=0
EC00239=0
EC00240=0
EC00241=0
EC00242=0
EC00243=0
EC00244=0
EC00245=0
EC00246=0
EC00247=0
EC00248=0
EC00249=0
EC00250=0
EC00251=0
EC00252=0
EC00253=0
EC00254=0
EC00255=0
EC00256=0
EC00257=0
EC00258=0
EC00259=0
EC00260=0
EC00261=0
EC00262=0
EC00263=0
EC00264=0
EC00265=0
EC00266=0
EC00267=0
EC00268=0
EC00269=0
EC00270=0
EC00271=0
EC00272=0
EC00273=0
EC00274=0
EC00275=0
EC00276=0
EC00277=0
EC00278=0
EC00279=0
EC00280=0
EC00281=0
EC00282=0
EC00283=0
EC00284=0
EC00285=0
EC00286=0
EC00287=0
EC00288=0
EC00289=0
EC00290=0
EC00291=0
EC00292=0
EC00293=0
EC00294=0
EC00295=0
EC00296=0
EC00297=0
EC00298=0
EC00299=0
EC00300=0
EC00301=0
EC00302=0
EC00303=0
EC00304=0
EC00305=0
EC00306=0
EC00307=0
EC00308=0
EC00309=0
EC00310=0
EC00311=0
EC00312=0
EC00313=0
EC00314=0
EC00315=0
EC00316=0
EC00317=0
EC00318=0
EC00319=90112.0
EC00320=90112.0
EC00321=90112.0
EC00322=90112.0
EC00323=90112.0
EC00324=90112.0
EC00325=90112.0
EC00326=90112.0
EC00327=90112.0
EC00328=90112.0
EC00329=90112.0
EC00330=90112.0
EC00331=90112.0
EC00332=90112.0
EC00333=274432.0
EC00334=274432.0
EC00335=274432.0
EC00336=274432.0
EC00337=274432.0
EC00338=274432.0
EC00339=274432.0
EC00340=274432.0
EC00341=274432.0
EC00342=274432.0
EC00343=274432.0
EC00344=274432.0
EC00345=274432.0
EC00346=274432.0
EC00347=277504.0
EC00348=277504.0
EC00349=277504.0
EC00350=277504.0
EC00351=277504.0
EC00352=277504.0
EC00353=277504.0
EC00354=277504.0
EC00355=277504.0
EC00356=277504.0
EC00357=277504.0
EC00358=277504.0
EC00359=277504.0
EC00360=277504.0
EC00361=277504.0
EC00362=277504.0
EC00363=277504.0
EC00364=277504.0
EC00365=277504.0
EC00366=277504.0
EC00367=277504.0
EC00368=277504.0
EC00369=277504.0
EC00370=277504.0
EC00371=277504.0
EC00372=277504.0
EC00373=277504.0
EC00374=277504.0
EC00375=277504.0
EC00376=277504.0
EC00377=277504.0
EC00378=277504.0
EC00379=277504.0
EC00380=277504.0
EC00381=277504.0
EC00382=277504.0
EC00383=277504.0
EC00384=277504.0
EC00385=277504.0
EC00386=277504.0
EC00387=277504.0
EC00388=277504.0
EC00389=277504.0
EC00390=277504.0
EC00391=277504.0
EC00392=277504.0
EC00393=277504.0
EC00394=277504.0
EC00395=277504.0
EC00396=277504.0
EC00397=277504.0
EC00398=277504.0
EC00399=277504.0
EC00400=277504.0
EC00401=277504.0
EC00402=277504.0
EC00403=277504.0
EC00404=277504.0
EC00405=277504.0
EC00406=277504.0
EC00407=277504.0
EC00408=277504.0
EC00409=277504.0
EC00410=277504.0
EC00411=277504.0
EC00412=277504.0
EC00413=277504.0
EC00414=277504.0
EC00415=277504.0
EC00416=277504.0
EC00417=277504.0
EC00418=277504.0
EC00419=277504.0
EC00420=277504.0
EC00421=277504.0
EC00422=277504.0
EC00423=277504.0
EC00424=277504.0
EC00425=277504.0
EC00426=277504.0
EC00427=277504.0
EC00428=277504.0
EC00429=277504.0
EC00430=277504.0
EC00431=277504.0
EC00432=277504.0
EC00433=277504.0
EC00434=277504.0
EC00435=277504.0
EC00436=277504.0
EC00437=277504.0
EC00438=277504.0
EC00439=277504.0
EC00440=277504.0
EC00441=277504.0
EC00442=277504.0
EC00443=277504.0
EC00444=277504.0
EC00445=277504.0
EC00446=277504.0
EC00447=277504.0
EC00448=277504.0
EC00449=277504.0
EC00450=277504.0
EC00451=277504.0
EC00452=277504.0
EC00453=277504.0
EC00454=277504.0
EC00455=277504.0
EC00456=277504.0
EC00457=277504.0
EC00458=277504.0
EC00459=277504.0
EC00460=277504.0
EC00461=277504.0
EC00462=277504.0
EC00463=277504.0
EC00464=277504.0
EC00465=277504.0
EC00466=277504.0
EC00467=277504.0
EC00468=277504.0
EC00469=277504.0
EC00470=277504.0
EC00471=277504.0
EC00472=277504.0
EC00473=277504.0
EC00474=277504.0
EC00475=277504.0
EC00476=277504.0
EC00477=277504.0
EC00478=277504.0
EC00479=277504.0
EC00480=277504.0
EC00481=277504.0
EC00482=277504.0
EC00483=277504.0
EC00484=277504.0
EC00485=277504.0
EC00486=277504.0
EC00487=277504.0
EC00488=277504.0
EC00489=277504.0
EC00490=277504.0
EC00491=277504.0
EC00492=277504.0
EC00493=277504.0
EC00494=277504.0
EC00495=277504.0
EC00496=277504.0
EC00497=277504.0
EC00498=277504.0
EC00499=277504.0
EC00500=277504.0
EC00501=277504.0
EC00502=277504.0
EC00503=277504.0
EC00504=277504.0
EC00505=277504.0
EC00506=277504.0
EC00507=277504.0
EC00508=277504.0
EC00509=277504.0
EC00510=277504.0
EC00511=277504.0
EC00512=277504.0
EC00513=277504.0
EC00514=277504.0
EC00515=277504.0
EC00516=277504.0
EC00517=277504.0
EC00518=277504.0
EC00519=277504.0
EC00520=277504.0
EC00521=277504.0
EC00522=277504.0
EC00523=277504.0
EC00524=277504.0
EC00525=277504.0
EC00526=277504.0
EC00527=277504.0
EC00528=277504.0
EC00529=277504.0
EC00530=277504.0
EC00531=277504.0
EC00532=277504.0
EC00533=277504.0
EC00534=277504.0
EC00535=277504.0
EC00536=277504.0
EC00537=277504.0
EC00538=277504.0
EC00539=277504.0
EC00540=277504.0
EC00541=277504.0
EC00542=277504.0
EC00543=277504.0
EC00544=277504.0
EC00545=277504.0
EC00546=277504.0
EC00547=277504.0
EC00548=277504.0
EC00549=277504.0
EC00550=277504.0
EC00551=277504.0
EC00552=277504.0
EC00553=277504.0
EC00554=277504.0
EC00555=277504.0
EC00556=277504.0
EC00557=277504.0
EC00558=277504.0
EC00559=277504.0
EC00560=277504.0
EC00561=277504.0
EC00562=277504.0
EC00563=277504.0
EC00564=277504.0
EC00565=277504.0
EC00566=277504.0
EC00567=277504.0
EC00568=277504.0
EC00569=277504.0
EC00570=277504.0
EC00571=277504.0
EC00572=277504.0
EC00573=277504.0
EC00574=277504.0
EC00575=277504.0
EC00576=277504.0
EC00577=277504.0
EC00578=277504.0
EC00579=277504.0
EC00580=277504.0
EC00581=277504.0
EC00582=277504.0
EC00583=277504.0
EC00584=277504.0
EC00585=277504.0
EC00586=277504.0
EC00587=277504.0
EC00588=277504.0
EC00589=277504.0
EC00590=277504.0
EC00591=277504.0
EC00592=277504.0
EC00593=277504.0
EC00594=277504.0
EC00595=277504.0
EC00596=277504.0
EC00597=277504.0
EC00598=367616.0
EC00599=367616.0
EC00600=367616.0
EC00601=367616.0
EC00602=367616.0
EC00603=367616.0
EC00604=367616.0
EC00605=367616.0
EC00606=367616.0
EC00607=367616.0
EC00608=367616.0
EC00609=367616.0
EC00610=367616.0
EC00611=367616.0
EC00612=367616.0
EC00613=367616.0
EC00614=367616.0
EC00615=367616.0
//INST
///DATE 2023/07/21 13:26
///ATTR SC,RW,RJ
////FRAME BASE
///GROUP1 RB1,ST1
NOP
MOVJ P009 EX000 VJ=15.00
MOVJ C00000 EC00000 VJ=15.0
CALL JOB:SPYON
MOVL C00001 EC00001 V=150
MOVL C00002 EC00002 V=150
MOVL C00003 EC00003 V=150
MOVL C00004 EC00004 V=150
MOVL C00005 EC00005 V=150
MOVL C00006 EC00006 V=150
MOVL C00007 EC00007 V=150
MOVL C00008 EC00008 V=150
MOVL C00009 EC00009 V=150
MOVL C00010 EC00010 V=150
MOVL C00011 EC00011 V=150
MOVL C00012 EC00012 V=150
MOVL C00013 EC00013 V=150
MOVL C00014 EC00014 V=150
MOVL C00015 EC00015 V=150
MOVL C00016 EC00016 V=150
MOVL C00017 EC00017 V=150
MOVL C00018 EC00018 V=150
MOVL C00019 EC00019 V=150
MOVL C00020 EC00020 V=150
MOVL C00021 EC00021 V=150
MOVL C00022 EC00022 V=150
MOVL C00023 EC00023 V=150
MOVL C00024 EC00024 V=150
MOVL C00025 EC00025 V=150
MOVL C00026 EC00026 V=150
MOVL C00027 EC00027 V=150
MOVL C00028 EC00028 V=150
MOVL C00029 EC00029 V=150
MOVL C00030 EC00030 V=150
MOVL C00031 EC00031 V=150
MOVL C00032 EC00032 V=150
MOVL C00033 EC00033 V=150
MOVL C00034 EC00034 V=150
MOVL C00035 EC00035 V=150
MOVL C00036 EC00036 V=150
MOVL C00037 EC00037 V=150
MOVL C00038 EC00038 V=150
MOVL C00039 EC00039 V=150
MOVL C00040 EC00040 V=150
MOVL C00041 EC00041 V=150
MOVL C00042 EC00042 V=150
MOVL C00043 EC00043 V=150
MOVL C00044 EC00044 V=150
MOVL C00045 EC00045 V=150
MOVL C00046 EC00046 V=150
MOVL C00047 EC00047 V=150
MOVL C00048 EC00048 V=150
MOVL C00049 EC00049 V=150
MOVL C00050 EC00050 V=150
MOVL C00051 EC00051 V=150
MOVL C00052 EC00052 V=150
MOVL C00053 EC00053 V=150
MOVL C00054 EC00054 V=150
MOVL C00055 EC00055 V=150
MOVL C00056 EC00056 V=150
MOVL C00057 EC00057 V=150
MOVL C00058 EC00058 V=150
MOVL C00059 EC00059 V=150
MOVL C00060 EC00060 V=150
MOVL C00061 EC00061 V=150
MOVL C00062 EC00062 V=150
MOVL C00063 EC00063 V=150
MOVL C00064 EC00064 V=150
MOVL C00065 EC00065 V=150
MOVL C00066 EC00066 V=150
MOVL C00067 EC00067 V=150
MOVL C00068 EC00068 V=150
MOVL C00069 EC00069 V=150
MOVL C00070 EC00070 V=150
MOVL C00071 EC00071 V=150
MOVL C00072 EC00072 V=150
MOVL C00073 EC00073 V=150
MOVL C00074 EC00074 V=150
MOVL C00075 EC00075 V=150
MOVL C00076 EC00076 V=150
MOVL C00077 EC00077 V=150
MOVL C00078 EC00078 V=150
MOVL C00079 EC00079 V=150
MOVL C00080 EC00080 V=150
MOVL C00081 EC00081 V=150
MOVL C00082 EC00082 V=150
MOVL C00083 EC00083 V=150
MOVL C00084 EC00084 V=150
MOVL C00085 EC00085 V=150
MOVL C00086 EC00086 V=150
MOVL C00087 EC00087 V=150
MOVL C00088 EC00088 V=150
MOVL C00089 EC00089 V=150
MOVL C00090 EC00090 V=150
MOVL C00091 EC00091 V=150
MOVL C00092 EC00092 V=150
MOVL C00093 EC00093 V=150
MOVL C00094 EC00094 V=150
MOVL C00095 EC00095 V=150
MOVL C00096 EC00096 V=150
MOVL C00097 EC00097 V=150
MOVL C00098 EC00098 V=150
MOVL C00099 EC00099 V=150
MOVL C00100 EC00100 V=150
MOVL C00101 EC00101 V=150
MOVL C00102 EC00102 V=150
MOVL C00103 EC00103 V=150
MOVL C00104 EC00104 V=150
MOVL C00105 EC00105 V=150
MOVL C00106 EC00106 V=150
MOVL C00107 EC00107 V=150
MOVL C00108 EC00108 V=150
MOVL C00109 EC00109 V=150
MOVL C00110 EC00110 V=150
MOVL C00111 EC00111 V=150
MOVL C00112 EC00112 V=150
MOVL C00113 EC00113 V=150
MOVL C00114 EC00114 V=150
MOVL C00115 EC00115 V=150
MOVL C00116 EC00116 V=150
MOVL C00117 EC00117 V=150
MOVL C00118 EC00118 V=150
MOVL C00119 EC00119 V=150
MOVL C00120 EC00120 V=150
MOVL C00121 EC00121 V=150
MOVL C00122 EC00122 V=150
MOVL C00123 EC00123 V=150
MOVL C00124 EC00124 V=150
MOVL C00125 EC00125 V=150
MOVL C00126 EC00126 V=150
MOVL C00127 EC00127 V=150
MOVL C00128 EC00128 V=150
MOVL C00129 EC00129 V=150
MOVL C00130 EC00130 V=150
MOVL C00131 EC00131 V=150
MOVL C00132 EC00132 V=150
MOVL C00133 EC00133 V=150
MOVL C00134 EC00134 V=150
MOVL C00135 EC00135 V=150
MOVL C00136 EC00136 V=150
MOVL C00137 EC00137 V=150
MOVL C00138 EC00138 V=150
MOVL C00139 EC00139 V=150
MOVL C00140 EC00140 V=150
MOVL C00141 EC00141 V=150
MOVL C00142 EC00142 V=150
MOVL C00143 EC00143 V=150
MOVL C00144 EC00144 V=150
MOVL C00145 EC00145 V=150
MOVL C00146 EC00146 V=150
MOVL C00147 EC00147 V=150
MOVL C00148 EC00148 V=150
MOVL C00149 EC00149 V=150
MOVL C00150 EC00150 V=150
MOVL C00151 EC00151 V=150
MOVL C00152 EC00152 V=150
MOVL C00153 EC00153 V=150
MOVL C00154 EC00154 V=150
MOVL C00155 EC00155 V=150
MOVL C00156 EC00156 V=150
MOVL C00157 EC00157 V=150
MOVL C00158 EC00158 V=150
MOVL C00159 EC00159 V=150
MOVL C00160 EC00160 V=150
MOVL C00161 EC00161 V=150
MOVL C00162 EC00162 V=150
MOVL C00163 EC00163 V=150
MOVL C00164 EC00164 V=150
MOVL C00165 EC00165 V=150
MOVL C00166 EC00166 V=150
MOVL C00167 EC00167 V=150
MOVL C00168 EC00168 V=150
MOVL C00169 EC00169 V=150
MOVL C00170 EC00170 V=150
MOVL C00171 EC00171 V=150
MOVL C00172 EC00172 V=150
MOVL C00173 EC00173 V=150
MOVL C00174 EC00174 V=150
MOVL C00175 EC00175 V=150
MOVL C00176 EC00176 V=150
MOVL C00177 EC00177 V=150
MOVL C00178 EC00178 V=150
MOVL C00179 EC00179 V=150
MOVL C00180 EC00180 V=150
MOVL C00181 EC00181 V=150
MOVL C00182 EC00182 V=150
MOVL C00183 EC00183 V=150
MOVL C00184 EC00184 V=150
MOVL C00185 EC00185 V=150
MOVL C00186 EC00186 V=150
MOVL C00187 EC00187 V=150
MOVL C00188 EC00188 V=150
MOVL C00189 EC00189 V=150
MOVL C00190 EC00190 V=150
MOVL C00191 EC00191 V=150
MOVL C00192 EC00192 V=150
MOVL C00193 EC00193 V=150
MOVL C00194 EC00194 V=150
MOVL C00195 EC00195 V=150
MOVL C00196 EC00196 V=150
MOVL C00197 EC00197 V=150
MOVL C00198 EC00198 V=150
MOVL C00199 EC00199 V=150
MOVL C00200 EC00200 V=150
MOVL C00201 EC00201 V=150
MOVL C00202 EC00202 V=150
MOVL C00203 EC00203 V=150
MOVL C00204 EC00204 V=150
MOVL C00205 EC00205 V=150
MOVL C00206 EC00206 V=150
MOVL C00207 EC00207 V=150
MOVL C00208 EC00208 V=150
MOVL C00209 EC00209 V=150
MOVL C00210 EC00210 V=150
MOVL C00211 EC00211 V=150
MOVL C00212 EC00212 V=150
MOVL C00213 EC00213 V=150
MOVL C00214 EC00214 V=150
MOVL C00215 EC00215 V=150
MOVL C00216 EC00216 V=150
MOVL C00217 EC00217 V=150
MOVL C00218 EC00218 V=150
MOVL C00219 EC00219 V=150
MOVL C00220 EC00220 V=150
MOVL C00221 EC00221 V=150
MOVL C00222 EC00222 V=150
MOVL C00223 EC00223 V=150
MOVL C00224 EC00224 V=150
MOVL C00225 EC00225 V=150
MOVL C00226 EC00226 V=150
MOVL C00227 EC00227 V=150
MOVL C00228 EC00228 V=150
MOVL C00229 EC00229 V=150
MOVL C00230 EC00230 V=150
MOVL C00231 EC00231 V=150
MOVL C00232 EC00232 V=150
MOVL C00233 EC00233 V=150
MOVL C00234 EC00234 V=150
MOVL C00235 EC00235 V=150
MOVL C00236 EC00236 V=150
MOVL C00237 EC00237 V=150
MOVL C00238 EC00238 V=150
MOVL C00239 EC00239 V=150
MOVL C00240 EC00240 V=150
MOVL C00241 EC00241 V=150
MOVL C00242 EC00242 V=150
MOVL C00243 EC00243 V=150
MOVL C00244 EC00244 V=150
MOVL C00245 EC00245 V=150
MOVL C00246 EC00246 V=150
MOVL C00247 EC00247 V=150
MOVL C00248 EC00248 V=150
MOVL C00249 EC00249 V=150
MOVL C00250 EC00250 V=150
MOVL C00251 EC00251 V=150
MOVL C00252 EC00252 V=150
MOVL C00253 EC00253 V=150
MOVL C00254 EC00254 V=150
MOVL C00255 EC00255 V=150
MOVL C00256 EC00256 V=150
MOVL C00257 EC00257 V=150
MOVL C00258 EC00258 V=150
MOVL C00259 EC00259 V=150
MOVL C00260 EC00260 V=150
MOVL C00261 EC00261 V=150
MOVL C00262 EC00262 V=150
MOVL C00263 EC00263 V=150
MOVL C00264 EC00264 V=150
MOVL C00265 EC00265 V=150
MOVL C00266 EC00266 V=150
MOVL C00267 EC00267 V=150
MOVL C00268 EC00268 V=150
MOVL C00269 EC00269 V=150
MOVL C00270 EC00270 V=150
MOVL C00271 EC00271 V=150
MOVL C00272 EC00272 V=150
MOVL C00273 EC00273 V=150
MOVL C00274 EC00274 V=150
MOVL C00275 EC00275 V=150
MOVL C00276 EC00276 V=150
MOVL C00277 EC00277 V=150
MOVL C00278 EC00278 V=150
MOVL C00279 EC00279 V=150
MOVL C00280 EC00280 V=150
MOVL C00281 EC00281 V=150
MOVL C00282 EC00282 V=150
MOVL C00283 EC00283 V=150
MOVL C00284 EC00284 V=150
MOVL C00285 EC00285 V=150
MOVL C00286 EC00286 V=150
MOVL C00287 EC00287 V=150
MOVL C00288 EC00288 V=150
MOVL C00289 EC00289 V=150
MOVL C00290 EC00290 V=150
MOVL C00291 EC00291 V=150
MOVL C00292 EC00292 V=150
MOVL C00293 EC00293 V=150
MOVL C00294 EC00294 V=150
MOVL C00295 EC00295 V=150
MOVL C00296 EC00296 V=150
MOVL C00297 EC00297 V=150
MOVL C00298 EC00298 V=150
MOVL C00299 EC00299 V=150
MOVL C00300 EC00300 V=150
MOVL C00301 EC00301 V=150
MOVL C00302 EC00302 V=150
MOVL C00303 EC00303 V=150
MOVL C00304 EC00304 V=150
MOVL C00305 EC00305 V=150
MOVL C00306 EC00306 V=150
MOVL C00307 EC00307 V=150
MOVL C00308 EC00308 V=150
MOVL C00309 EC00309 V=150
MOVL C00310 EC00310 V=150
MOVL C00311 EC00311 V=150
MOVL C00312 EC00312 V=150
MOVL C00313 EC00313 V=150
MOVL C00314 EC00314 V=150
MOVL C00315 EC00315 V=150
MOVL C00316 EC00316 V=150
MOVL C00317 EC00317 V=150
MOVL C00318 EC00318 V=150
CALL JOB:SPYOF
MOVJ P009 VJ=15.00
MOVJ C00319 EC00319 VJ=15.0
CALL JOB:SPYON
MOVL C00320 EC00320 V=150
MOVL C00321 EC00321 V=150
MOVL C00322 EC00322 V=150
MOVL C00323 EC00323 V=150
MOVL C00324 EC00324 V=150
MOVL C00325 EC00325 V=150
MOVL C00326 EC00326 V=150
MOVL C00327 EC00327 V=150
MOVL C00328 EC00328 V=150
MOVL C00329 EC00329 V=150
MOVL C00330 EC00330 V=150
MOVL C00331 EC00331 V=150
MOVL C00332 EC00332 V=150
CALL JOB:SPYOF
MOVJ P009 VJ=15.00
MOVJ C00333 EC00333 VJ=15.0
CALL JOB:SPYON
MOVL C00334 EC00334 V=150
MOVL C00335 EC00335 V=150
MOVL C00336 EC00336 V=150
MOVL C00337 EC00337 V=150
MOVL C00338 EC00338 V=150
MOVL C00339 EC00339 V=150
MOVL C00340 EC00340 V=150
MOVL C00341 EC00341 V=150
MOVL C00342 EC00342 V=150
MOVL C00343 EC00343 V=150
MOVL C00344 EC00344 V=150
MOVL C00345 EC00345 V=150
MOVL C00346 EC00346 V=150
CALL JOB:SPYOF
MOVJ P009 VJ=15.00
MOVJ C00347 EC00347 VJ=15.0
CALL JOB:SPYON
MOVL C00348 EC00348 V=150
MOVL C00349 EC00349 V=150
MOVL C00350 EC00350 V=150
MOVL C00351 EC00351 V=150
MOVL C00352 EC00352 V=150
MOVL C00353 EC00353 V=150
MOVL C00354 EC00354 V=150
MOVL C00355 EC00355 V=150
MOVL C00356 EC00356 V=150
MOVL C00357 EC00357 V=150
MOVL C00358 EC00358 V=150
MOVL C00359 EC00359 V=150
MOVL C00360 EC00360 V=150
MOVL C00361 EC00361 V=150
MOVL C00362 EC00362 V=150
MOVL C00363 EC00363 V=150
MOVL C00364 EC00364 V=150
MOVL C00365 EC00365 V=150
MOVL C00366 EC00366 V=150
MOVL C00367 EC00367 V=150
MOVL C00368 EC00368 V=150
MOVL C00369 EC00369 V=150
MOVL C00370 EC00370 V=150
MOVL C00371 EC00371 V=150
MOVL C00372 EC00372 V=150
MOVL C00373 EC00373 V=150
MOVL C00374 EC00374 V=150
MOVL C00375 EC00375 V=150
MOVL C00376 EC00376 V=150
MOVL C00377 EC00377 V=150
MOVL C00378 EC00378 V=150
MOVL C00379 EC00379 V=150
MOVL C00380 EC00380 V=150
MOVL C00381 EC00381 V=150
MOVL C00382 EC00382 V=150
MOVL C00383 EC00383 V=150
MOVL C00384 EC00384 V=150
MOVL C00385 EC00385 V=150
MOVL C00386 EC00386 V=150
MOVL C00387 EC00387 V=150
MOVL C00388 EC00388 V=150
MOVL C00389 EC00389 V=150
MOVL C00390 EC00390 V=150
MOVL C00391 EC00391 V=150
MOVL C00392 EC00392 V=150
MOVL C00393 EC00393 V=150
MOVL C00394 EC00394 V=150
MOVL C00395 EC00395 V=150
MOVL C00396 EC00396 V=150
MOVL C00397 EC00397 V=150
MOVL C00398 EC00398 V=150
MOVL C00399 EC00399 V=150
MOVL C00400 EC00400 V=150
MOVL C00401 EC00401 V=150
MOVL C00402 EC00402 V=150
MOVL C00403 EC00403 V=150
MOVL C00404 EC00404 V=150
MOVL C00405 EC00405 V=150
MOVL C00406 EC00406 V=150
MOVL C00407 EC00407 V=150
MOVL C00408 EC00408 V=150
MOVL C00409 EC00409 V=150
MOVL C00410 EC00410 V=150
MOVL C00411 EC00411 V=150
MOVL C00412 EC00412 V=150
MOVL C00413 EC00413 V=150
MOVL C00414 EC00414 V=150
MOVL C00415 EC00415 V=150
MOVL C00416 EC00416 V=150
MOVL C00417 EC00417 V=150
MOVL C00418 EC00418 V=150
MOVL C00419 EC00419 V=150
MOVL C00420 EC00420 V=150
MOVL C00421 EC00421 V=150
MOVL C00422 EC00422 V=150
MOVL C00423 EC00423 V=150
MOVL C00424 EC00424 V=150
MOVL C00425 EC00425 V=150
MOVL C00426 EC00426 V=150
MOVL C00427 EC00427 V=150
MOVL C00428 EC00428 V=150
MOVL C00429 EC00429 V=150
MOVL C00430 EC00430 V=150
MOVL C00431 EC00431 V=150
MOVL C00432 EC00432 V=150
MOVL C00433 EC00433 V=150
MOVL C00434 EC00434 V=150
MOVL C00435 EC00435 V=150
MOVL C00436 EC00436 V=150
MOVL C00437 EC00437 V=150
MOVL C00438 EC00438 V=150
MOVL C00439 EC00439 V=150
MOVL C00440 EC00440 V=150
MOVL C00441 EC00441 V=150
MOVL C00442 EC00442 V=150
MOVL C00443 EC00443 V=150
MOVL C00444 EC00444 V=150
MOVL C00445 EC00445 V=150
MOVL C00446 EC00446 V=150
MOVL C00447 EC00447 V=150
MOVL C00448 EC00448 V=150
MOVL C00449 EC00449 V=150
MOVL C00450 EC00450 V=150
MOVL C00451 EC00451 V=150
MOVL C00452 EC00452 V=150
MOVL C00453 EC00453 V=150
MOVL C00454 EC00454 V=150
MOVL C00455 EC00455 V=150
MOVL C00456 EC00456 V=150
MOVL C00457 EC00457 V=150
MOVL C00458 EC00458 V=150
MOVL C00459 EC00459 V=150
MOVL C00460 EC00460 V=150
MOVL C00461 EC00461 V=150
MOVL C00462 EC00462 V=150
MOVL C00463 EC00463 V=150
MOVL C00464 EC00464 V=150
MOVL C00465 EC00465 V=150
MOVL C00466 EC00466 V=150
MOVL C00467 EC00467 V=150
MOVL C00468 EC00468 V=150
MOVL C00469 EC00469 V=150
MOVL C00470 EC00470 V=150
MOVL C00471 EC00471 V=150
MOVL C00472 EC00472 V=150
MOVL C00473 EC00473 V=150
MOVL C00474 EC00474 V=150
MOVL C00475 EC00475 V=150
MOVL C00476 EC00476 V=150
MOVL C00477 EC00477 V=150
MOVL C00478 EC00478 V=150
MOVL C00479 EC00479 V=150
MOVL C00480 EC00480 V=150
MOVL C00481 EC00481 V=150
MOVL C00482 EC00482 V=150
MOVL C00483 EC00483 V=150
MOVL C00484 EC00484 V=150
MOVL C00485 EC00485 V=150
MOVL C00486 EC00486 V=150
MOVL C00487 EC00487 V=150
MOVL C00488 EC00488 V=150
MOVL C00489 EC00489 V=150
MOVL C00490 EC00490 V=150
MOVL C00491 EC00491 V=150
MOVL C00492 EC00492 V=150
MOVL C00493 EC00493 V=150
MOVL C00494 EC00494 V=150
MOVL C00495 EC00495 V=150
MOVL C00496 EC00496 V=150
MOVL C00497 EC00497 V=150
MOVL C00498 EC00498 V=150
MOVL C00499 EC00499 V=150
MOVL C00500 EC00500 V=150
MOVL C00501 EC00501 V=150
MOVL C00502 EC00502 V=150
MOVL C00503 EC00503 V=150
MOVL C00504 EC00504 V=150
MOVL C00505 EC00505 V=150
MOVL C00506 EC00506 V=150
MOVL C00507 EC00507 V=150
MOVL C00508 EC00508 V=150
MOVL C00509 EC00509 V=150
MOVL C00510 EC00510 V=150
MOVL C00511 EC00511 V=150
MOVL C00512 EC00512 V=150
MOVL C00513 EC00513 V=150
MOVL C00514 EC00514 V=150
MOVL C00515 EC00515 V=150
MOVL C00516 EC00516 V=150
MOVL C00517 EC00517 V=150
MOVL C00518 EC00518 V=150
MOVL C00519 EC00519 V=150
MOVL C00520 EC00520 V=150
MOVL C00521 EC00521 V=150
MOVL C00522 EC00522 V=150
MOVL C00523 EC00523 V=150
MOVL C00524 EC00524 V=150
MOVL C00525 EC00525 V=150
MOVL C00526 EC00526 V=150
MOVL C00527 EC00527 V=150
MOVL C00528 EC00528 V=150
MOVL C00529 EC00529 V=150
MOVL C00530 EC00530 V=150
MOVL C00531 EC00531 V=150
MOVL C00532 EC00532 V=150
MOVL C00533 EC00533 V=150
MOVL C00534 EC00534 V=150
MOVL C00535 EC00535 V=150
MOVL C00536 EC00536 V=150
MOVL C00537 EC00537 V=150
MOVL C00538 EC00538 V=150
MOVL C00539 EC00539 V=150
MOVL C00540 EC00540 V=150
MOVL C00541 EC00541 V=150
MOVL C00542 EC00542 V=150
MOVL C00543 EC00543 V=150
MOVL C00544 EC00544 V=150
MOVL C00545 EC00545 V=150
MOVL C00546 EC00546 V=150
MOVL C00547 EC00547 V=150
MOVL C00548 EC00548 V=150
MOVL C00549 EC00549 V=150
MOVL C00550 EC00550 V=150
MOVL C00551 EC00551 V=150
MOVL C00552 EC00552 V=150
MOVL C00553 EC00553 V=150
MOVL C00554 EC00554 V=150
MOVL C00555 EC00555 V=150
MOVL C00556 EC00556 V=150
MOVL C00557 EC00557 V=150
MOVL C00558 EC00558 V=150
MOVL C00559 EC00559 V=150
MOVL C00560 EC00560 V=150
MOVL C00561 EC00561 V=150
MOVL C00562 EC00562 V=150
MOVL C00563 EC00563 V=150
MOVL C00564 EC00564 V=150
MOVL C00565 EC00565 V=150
MOVL C00566 EC00566 V=150
MOVL C00567 EC00567 V=150
MOVL C00568 EC00568 V=150
MOVL C00569 EC00569 V=150
MOVL C00570 EC00570 V=150
MOVL C00571 EC00571 V=150
MOVL C00572 EC00572 V=150
MOVL C00573 EC00573 V=150
MOVL C00574 EC00574 V=150
MOVL C00575 EC00575 V=150
MOVL C00576 EC00576 V=150
MOVL C00577 EC00577 V=150
MOVL C00578 EC00578 V=150
MOVL C00579 EC00579 V=150
MOVL C00580 EC00580 V=150
MOVL C00581 EC00581 V=150
MOVL C00582 EC00582 V=150
MOVL C00583 EC00583 V=150
MOVL C00584 EC00584 V=150
MOVL C00585 EC00585 V=150
MOVL C00586 EC00586 V=150
MOVL C00587 EC00587 V=150
MOVL C00588 EC00588 V=150
MOVL C00589 EC00589 V=150
MOVL C00590 EC00590 V=150
MOVL C00591 EC00591 V=150
MOVL C00592 EC00592 V=150
MOVL C00593 EC00593 V=150
MOVL C00594 EC00594 V=150
MOVL C00595 EC00595 V=150
MOVL C00596 EC00596 V=150
MOVL C00597 EC00597 V=150
CALL JOB:SPYOF
MOVJ P009 VJ=15.00
MOVJ C00598 EC00598 VJ=15.0
CALL JOB:SPYON
MOVL C00599 EC00599 V=150
MOVL C00600 EC00600 V=150
MOVL C00601 EC00601 V=150
MOVL C00602 EC00602 V=150
MOVL C00603 EC00603 V=150
MOVL C00604 EC00604 V=150
MOVL C00605 EC00605 V=150
MOVL C00606 EC00606 V=150
MOVL C00607 EC00607 V=150
MOVL C00608 EC00608 V=150
MOVL C00609 EC00609 V=150
MOVL C00610 EC00610 V=150
MOVL C00611 EC00611 V=150
MOVL C00612 EC00612 V=150
MOVL C00613 EC00613 V=150
MOVL C00614 EC00614 V=150
MOVL C00615 EC00615 V=150
CALL JOB:SPYOF
MOVJ P009 VJ=15.00
END
